(* CODESYS project Reguleringsundervisning.project

Project tree, tasks and I/O mapping:
  Device : CODESYS Control Win V3 x64, 3S - Smart Software Solutions GmbH, version 3.5.16.20
    application Application
      libraries: Standard, * (System); VisuDialogs, * (System); Util, * (System); Gand Funksjonsbibliotek, 1.1 (Gand VGS)
      task MainTask (cyclic, interval t#1ms, priority 1) calls PLC_PRG
      task ReguTask (cyclic, interval t#20ms, priority 1) calls TilbakekobletRegulering, Reguleringsprogram
      task AlarmManagerTask (cyclic, interval 50 ms, priority 31) calls AlarmManager.Alarm_Prg
      task VISU_TASK (cyclic, interval 50 ms, priority 31) calls VisuElems.Visu_Prg
      program PLC_PRG [FBD]
      Level3/
        visualisation Level3_RepOppgave_ZogN
        visualisation Level3_TilbakekobletRegulering
      TilbakekobletRegulering/
        program TilbakekobletRegulering [FBD]
        program Reguleringsprogram [FBD]
      visualisation FlytteEksempel
      global variables GVL
      Level2/
        visualisation Level2_LIC01
      Level1/
        visualisation Level1
      Level4/
        visualisation Level4_TilbakekobletRegulering_Optimalisering
      visualisation Hovedmeny
      Skogestadsmetode/
        visualisation Level3_SkogestadsMetode
        visualisation Level3_SkogestadsMetode_Nav
        visualisation Level3_SkogestadsMetode_tab1
        visualisation Level3_SkogestadsMetode_tab2
        visualisation Level3_SkogestadsMetode_tab3
        visualisation Level3_SkogestadsMetode_tab4
      FacePlates/
        visualisation Faceplate_template
        visualisation RepOppgave_FacePlate
        visualisation ZieglerNicholsSvinge1
        visualisation ZieglerNicholsSvinge2
        visualisation ZieglerNicholsSvinge3
        visualisation ZieglerNicholsSvinge4
        visualisation ZieglerNicholsSvinge5
        visualisation ZieglerNicholsSvinge6
        visualisation ZieglerNicholsSvinge7
      image pool ImagePool
      Dialogs/
        visualisation LIC01_settings
      program Belastningsim [ST]
      Symbols
      Alarm Configuration
        alarm class Error (priority 10, acknowledge REP_ACK)
        alarm class Warning (priority 30, acknowledge REP_ACK)
        alarm class Info (priority 100, acknowledge REP)
        AlarmStorage
        text list AlarmGroup1
        alarm group AlarmGroup1
            0 [Warning]: Comparison Greater, ExpressionToCompare 80, Hysteresis 5, Expression TilbakekobletRegulering.LOOP01.rPV - "Nivå høyt i vanntank"
  text list GlobalTextList
  5ce3da45-db07-42e7-a21c-a00fff4ed8f6|C:\Users\fred-olav\Pictures\Screenshots\Prosessdata.PNG
  5ce3da45-db07-42e7-a21c-a00fff4ed8f6|C:\Users\fred-olav\Pictures\Screenshots\IntProsess.PNG
  5ce3da45-db07-42e7-a21c-a00fff4ed8f6|C:\Users\Mosdal\Pictures\Formler tidskonsstant.PNG
  5ce3da45-db07-42e7-a21c-a00fff4ed8f6|C:\Users\Mosdal\Pictures\intprosess.png
  5ce3da45-db07-42e7-a21c-a00fff4ed8f6|C:\Users\Mosdal\Pictures\Formler intpros.PNG
  5ce3da45-db07-42e7-a21c-a00fff4ed8f6|C:\Users\fred-olav\Pictures\Screenshots\Formler selvregulerende.PNG
  5ce3da45-db07-42e7-a21c-a00fff4ed8f6|C:\Users\fred-olav\Pictures\Screenshots\Skjermbilde.JPG
  5ce3da45-db07-42e7-a21c-a00fff4ed8f6|C:\Users\fred-olav\Pictures\Screenshots\Formler integrerende.PNG
*)

// Device/Application/GVL
VAR_GLOBAL
	TLX:INT :=0;
	TLY:INT :=0;
	BRX:INT :=0;
	BRY:INT :=0;
	
	iSelector :INT:=1;
	
	LOOP02: Gand.Loop_CAS :=(rKp := 1.7, rTi := 10, Navn := 'LIC02', rTi_slave := 0.3);
	LOOP03: Gand.Loop_CAS := (rKp := -9.3, rTi := 15, Navn := 'Tank Nivå', rKp_slave := 0.444, rTi_slave := 2.25);
	LOOP04: Gand.Loop :=(Navn := 'Tank Nivå');
	
END_VAR

VAR_GLOBAL CONSTANT
	iMax_Pumps : INT :=10;
END_VAR

// Device/Application/PLC_PRG
PROGRAM PLC_PRG
VAR
	SP_U: BOOL;
	Verdi: REAL;
	SP: REAL;
	LLA: BOOL;
	HHA: BOOL;
	NormalShifte: REAL;
	MaxVerdi: REAL :=100;
	MinVerdi: REAL;
	HILV: REAL := 95;
	HHV: REAL :=90;
	HV: REAL := 80;
	NormalTop: REAL :=70;
	NormalBottom: REAL :=30;
	LV: REAL := 20;
	LLV: REAL :=10;
	LILV: REAL := 5;
END_VAR

// NETWORK 1

END_PROGRAM

// Device/Application/TilbakekobletRegulering/TilbakekobletRegulering
PROGRAM TilbakekobletRegulering
VAR
	Int_tids_prosess_0: Gand.Int_tids_prosess;
	Tank: Gand.Int_tids_prosess;
	LIC01: PID;
	LOOP01: Gand.Loop;
	
END_VAR
VAR_INPUT
	Belastning_LIC01: REAL :=50;
END_VAR

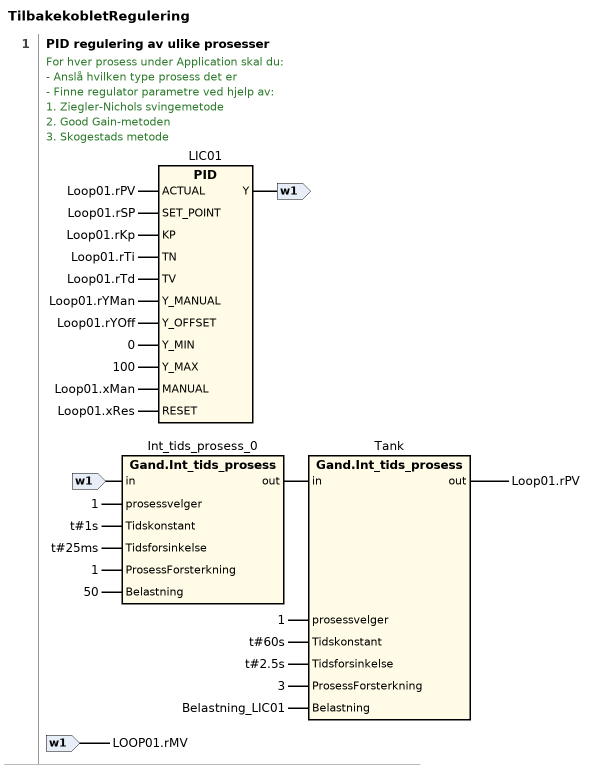
// NETWORK 1: PID regulering av ulike prosesser
// For hver prosess under Application skal du:
// - Anslå hvilken type prosess det er
// - Finne regulator parametre ved hjelp av:
// 	1. Ziegler-Nichols svingemetode
// 	2. Good Gain-metoden
// 	3. Skogestads metode
LIC01(
    ACTUAL := Loop01.rPV,
    SET_POINT := Loop01.rSP,
    KP := Loop01.rKp,
    TN := Loop01.rTi,
    TV := Loop01.rTd,
    Y_MANUAL := Loop01.rYMan,
    Y_OFFSET := Loop01.rYOff,
    Y_MIN := 0,
    Y_MAX := 100,
    MANUAL := Loop01.xMan,
    RESET := Loop01.xRes); // PID
Int_tids_prosess_0(
    in := LIC01.Y,
    prosessvelger := 1,
    Tidskonstant := t#1s,
    Tidsforsinkelse := t#25ms,
    ProsessForsterkning := 1,
    Belastning := 50); // Gand.Int_tids_prosess
Tank(
    in := Int_tids_prosess_0.out,
    prosessvelger := 1,
    Tidskonstant := t#60s,
    Tidsforsinkelse := t#2.5s,
    ProsessForsterkning := 3,
    Belastning := Belastning_LIC01); // Gand.Int_tids_prosess
Loop01.rPV := Tank.out;
LOOP01.rMV := LIC01.Y;

END_PROGRAM

// Device/Application/TilbakekobletRegulering/Reguleringsprogram
PROGRAM Reguleringsprogram
VAR
	PID01: PID;
	rSP_PID01: REAL :=50;
	rKP_PID01: REAL := 2;
	rTN_PID01: REAL := 2;
	rTV_PID01: REAL := 0;
	rYman_PID01: REAL := 20;
	rOff_PID01: REAL := 20;
	xMan_PID01: BOOL;
	xRes_PID01: BOOL;
	xLim_PID01: BOOL;
	xOvFlow_PID01: BOOL;
	Prosessnr: INT :=1;
	Prosess01: Gand.Prosess;
	
END_VAR
VAR_INPUT
	
END_VAR

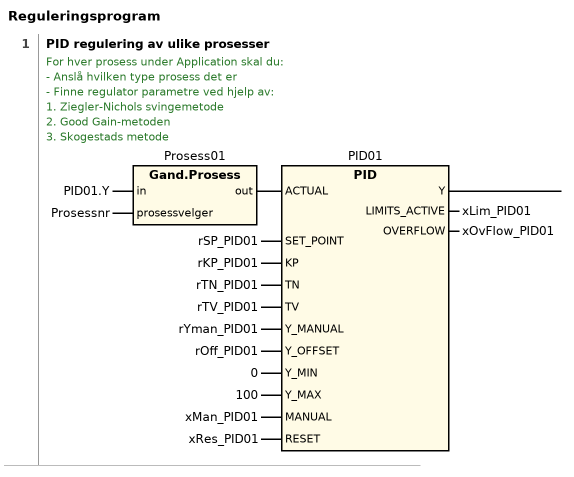
// NETWORK 1: PID regulering av ulike prosesser
// For hver prosess under Application skal du:
// - Anslå hvilken type prosess det er
// - Finne regulator parametre ved hjelp av:
// 	1. Ziegler-Nichols svingemetode
// 	2. Good Gain-metoden
// 	3. Skogestads metode
Prosess01(in := PID01.Y, prosessvelger := Prosessnr); // Gand.Prosess
PID01(
    ACTUAL := Prosess01.out,
    SET_POINT := rSP_PID01,
    KP := rKP_PID01,
    TN := rTN_PID01,
    TV := rTV_PID01,
    Y_MANUAL := rYman_PID01,
    Y_OFFSET := rOff_PID01,
    Y_MIN := 0,
    Y_MAX := 100,
    MANUAL := xMan_PID01,
    RESET := xRes_PID01,
    LIMITS_ACTIVE => xLim_PID01,
    OVERFLOW => xOvFlow_PID01); // PID

END_PROGRAM

// Device/Application/Belastningsim
PROGRAM Belastningsim
VAR
	step : INT :=1;
	i: INT;
	belastning: REAL := 50;
	timer1:TON := (PT := T#30S);
	Inntimer: BOOL :=FALSE;
END_VAR

CASE step OF
	1: 
	IF i < 100 THEN
		i:=i+1;
	ELSE
		belastning:=belastning+1;
		TilbakekobletRegulering.Belastning_LIC01:=belastning;
		i:=1;
		step:=step+1;
	END_IF
	2: 
	IF i < 100 THEN
		i:=i+1;
	ELSE
		belastning:=belastning+1;
		TilbakekobletRegulering.Belastning_LIC01:=belastning;
		i:=1;
		step:=step+1;
	END_IF
	3: 
	IF i < 100 THEN
		i:=i+1;
	ELSE
		belastning:=belastning+1;
		TilbakekobletRegulering.Belastning_LIC01:=belastning;
		i:=1;
		step:=step+1;
	END_IF
	4: 
	IF i < 100 THEN
		i:=i+1;
	ELSE
		belastning:=belastning+1;
		TilbakekobletRegulering.Belastning_LIC01:=belastning;
		i:=1;
		step:=step+1;
	END_IF
	5: 
	IF i < 100 THEN
		i:=i+1;
	ELSE
		belastning:=belastning+1;
		TilbakekobletRegulering.Belastning_LIC01:=belastning;
		i:=1;
		step:=step+1;
	END_IF
	6: 
	IF i < 100 THEN
		i:=i+1;
	ELSE
		belastning:=belastning+1;
		TilbakekobletRegulering.Belastning_LIC01:=belastning;
		i:=1;
		step:=step+1;
	END_IF
	7: 
	IF i < 100 THEN
		i:=i+1;
	ELSE
		belastning:=belastning+1;
		TilbakekobletRegulering.Belastning_LIC01:=belastning;
		i:=1;
		step:=step+1;
	END_IF
	8: 
	IF i < 100 THEN
		i:=i+1;
	ELSE
		belastning:=belastning+1;
		TilbakekobletRegulering.Belastning_LIC01:=belastning;
		i:=1;
		step:=step+1;
	END_IF
	9: 
	IF i < 100 THEN
		i:=i+1;
	ELSE
		belastning:=belastning+1;
		TilbakekobletRegulering.Belastning_LIC01:=belastning;
		i:=1;
		step:=step+1;
	END_IF
	10: 
	IF NOT Inntimer THEN
		
		IF i < 100 THEN
			i:=i+1;
		ELSE
			belastning:=belastning+1;
			TilbakekobletRegulering.Belastning_LIC01:=belastning;
			Inntimer:=TRUE;		
		END_IF
	ELSE
		IF timer1.Q THEN
		inntimer:=FALSE;
		 i:=1;
		step:=step+1;
		ELSE;
		END_IF
	END_IF
	timer1.IN:=inntimer;
	11: 
	IF i < 100 THEN
		i:=i+1;
	ELSE
		belastning:=belastning+1;
		TilbakekobletRegulering.Belastning_LIC01:=belastning;
		i:=1;
		step:=step+1;
	END_IF
	12: 
	IF i < 100 THEN
		i:=i+1;
	ELSE
		belastning:=belastning+1;
		TilbakekobletRegulering.Belastning_LIC01:=belastning;
		i:=1;
		step:=step+1;
	END_IF
	13: 
	IF i < 100 THEN
		i:=i+1;
	ELSE
		belastning:=belastning+1;
		TilbakekobletRegulering.Belastning_LIC01:=belastning;
		i:=1;
		step:=step+1;
	END_IF
	14: 
	IF i < 100 THEN
		i:=i+1;
	ELSE
		belastning:=belastning+1;
		TilbakekobletRegulering.Belastning_LIC01:=belastning;
		i:=1;
		step:=step+1;
		
	END_IF
	15: 
	IF i < 100 THEN
		i:=i+1;
	ELSE
		belastning:=belastning+1;
		TilbakekobletRegulering.Belastning_LIC01:=belastning;
		i:=1;
		step:=step+1;
	END_IF
	16: 
	IF i < 100 THEN
		i:=i+1;
	ELSE
		belastning:=belastning+1;
		TilbakekobletRegulering.Belastning_LIC01:=belastning;
		i:=1;
		step:=step+1;
	END_IF
	17: 
	IF i < 100 THEN
		i:=i+1;
	ELSE
		belastning:=belastning+1;
		TilbakekobletRegulering.Belastning_LIC01:=belastning;
		i:=1;
		step:=step+1;
	END_IF
	18: 
	IF i < 100 THEN
		i:=i+1;
	ELSE
		belastning:=belastning+1;
		TilbakekobletRegulering.Belastning_LIC01:=belastning;
		i:=1;
		step:=step+1;
	END_IF
	
END_CASE

END_PROGRAM

// Device/Application/Level4/Level4_TilbakekobletRegulering_Optimalisering
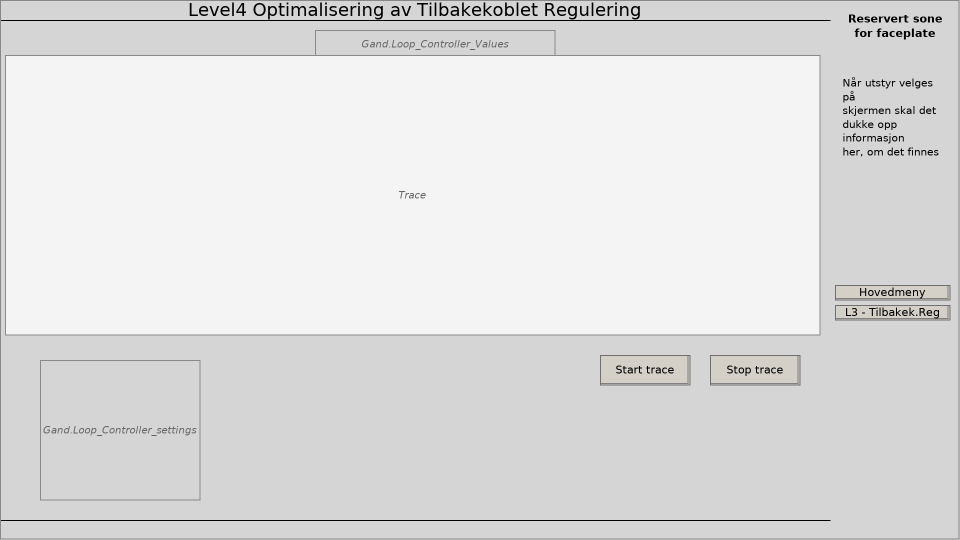
VISUALIZATION Level4_TilbakekobletRegulering_Optimalisering  // 960x540
VAR_IN_OUT
END_VAR
VAR
	bResetTrigger : BOOL;
	bStart : BOOL;
	bStop : BOOL;
	bStore : BOOL;
	sStoreFilename : STRING;
	bRestore : BOOL;
	sRestoreFilename : STRING;
END_VAR
    Frame (835,0 120x270)
        shows Faceplate_template()
        shows Navigation_template()
    Line (0,20) (830,20)
    Line (0,520) (830,520)
    Button (835,285 115x15), "Hovedmeny"
        OnMouseClick:  Assign=Hovedmeny, Type=Assignment
    Button (835,305 115x15), "L3 - Tilbakek.Reg"
        OnMouseClick:  Assign=Level3_TilbakekobletRegulering, Type=Assignment
    Label (0,0 830x20), "Level4 Optimalisering av Tilbakekoblet Regulering"
    Frame (40,360 160x140)
        shows Gand.Loop_Controller_settings(Local_data := TilbakekobletRegulering.LOOP01)
    Frame (315,30 240x28)
        shows Gand.Loop_Controller_Values(Local_data := TilbakekobletRegulering.LOOP01)
    Trace (5,55 815x280)
        p866368322: bStart
        p3851742229: bStop
    Button (600,355 90x30), "Start trace"
        toggle bStart
    Button (710,355 90x30), "Stop trace"
        toggle bStop
END_VISUALIZATION

// Device/Application/FlytteEksempel
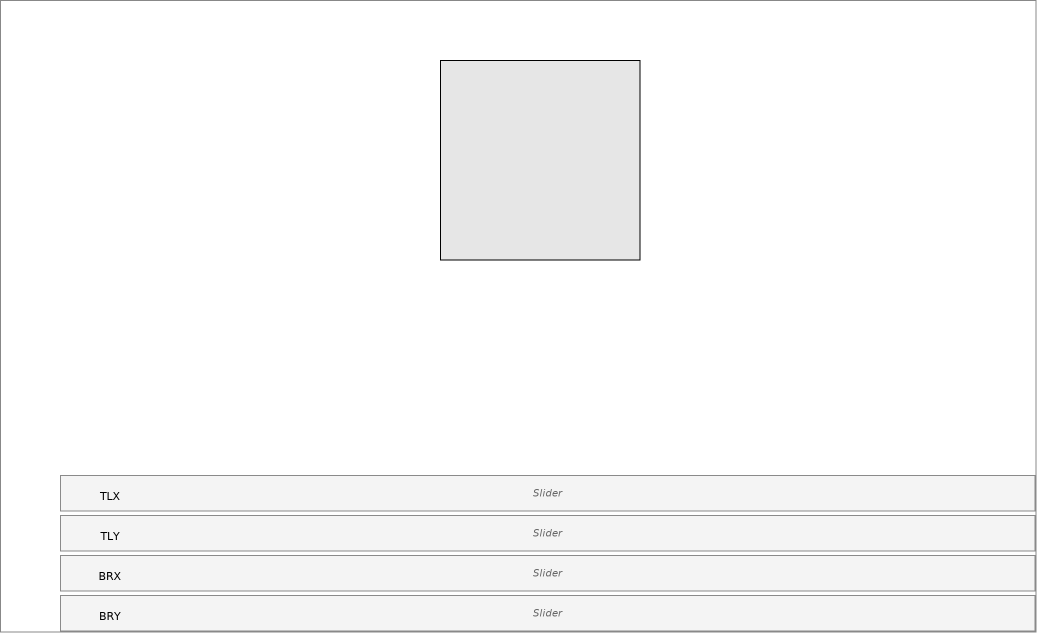
VISUALIZATION FlytteEksempel  // 1037x633
    Rectangle (440,60 200x200)
    Slider (60,475 975x36), variable: TLX, scale 0..100
    Slider (60,515 975x36), variable: TLY, scale 0..100
    Slider (60,555 975x36), variable: BRX, scale 0..100
    Slider (60,595 975x36), variable: BRY, scale 0..100
    Label (92,605 36x23), "BRY"
    Label (92,565 36x23), "BRX"
    Label (92,525 36x23), "TLY"
    Label (92,485 36x23), "TLX"
END_VISUALIZATION

// Device/Application/Level2/Level2_LIC01
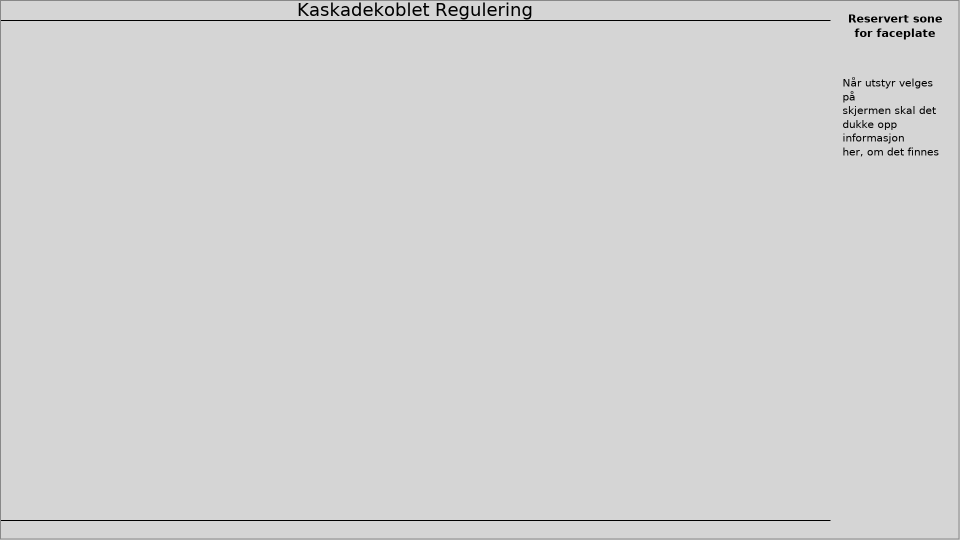
VISUALIZATION Level2_LIC01  // 960x540
VAR_IN_OUT
END_VAR
VAR
	bResetTrigger : BOOL;
	bStart : BOOL;
	bStop : BOOL;
	bStore : BOOL;
	sStoreFilename : STRING;
	bRestore : BOOL;
	sRestoreFilename : STRING;
END_VAR
    Frame (835,0 120x270)
        shows Faceplate_template()
        shows Navigation_template()
    Line (0,20) (830,20)
    Line (0,520) (830,520)
    Label (295,0 240x20), "Kaskadekoblet Regulering"
END_VISUALIZATION

// Device/Application/FacePlates/Faceplate_template
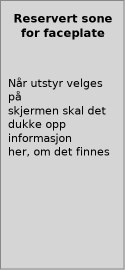
VISUALIZATION Faceplate_template  // 125x270
    Label (-12,11 150x30), "Reservert sone for faceplate"
    Label (5,75 115x85), "Når utstyr velges på skjermen skal det dukke opp informasjon her, om det finnes"
END_VISUALIZATION

// Device/Application/Hovedmeny
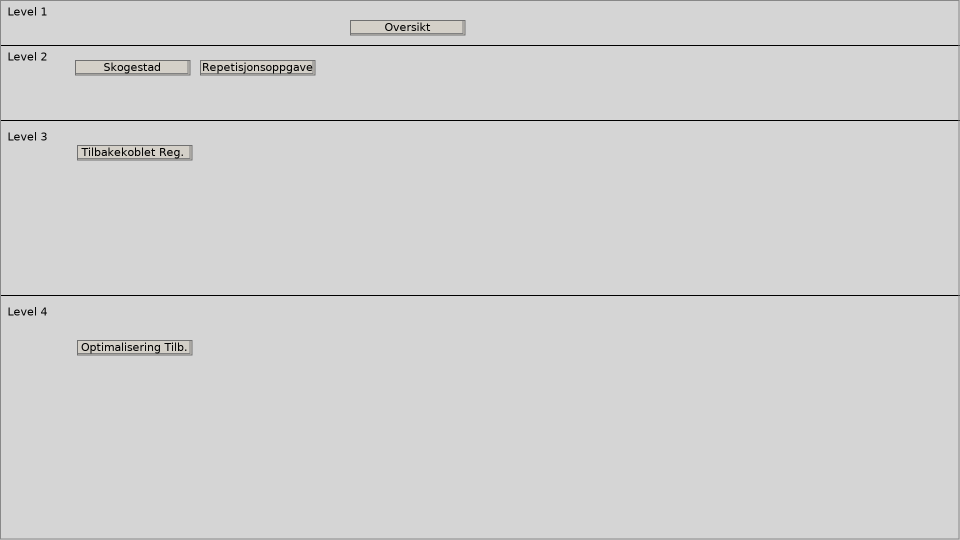
VISUALIZATION Hovedmeny  // 960x540
    Button (350,20 115x15), "Oversikt"
        OnMouseClick:  Assign=Level1, Type=Assignment
    Line (0,45) (960,45)
    Label (0,50 55x14), "Level 2"
    Label (0,130 55x14), "Level 3"
    Label (0,305 55x14), "Level 4"
    Label (0,5 55x14), "Level 1"
    Line (0,120) (960,120)
    Line (0,295) (960,295)
    Button (200,60 115x15), "Repetisjonsoppgave"
        OnMouseClick:  Assign=Level3_RepOppgave_ZogN, Type=Assignment
    Button (75,60 115x15), "Skogestad"
        OnMouseClick:  Assign=Level3_SkogestadsMetode, Type=Assignment
    Button (77,340 115x15), "Optimalisering Tilb."
        OnMouseClick:  Assign=Level4_TilbakekobletRegulering_Optimalisering, Type=Assignment
    Button (77,145 115x15), "Tilbakekoblet Reg."
        OnMouseClick:  Assign=Level3_TilbakekobletRegulering, Type=Assignment
END_VISUALIZATION

// Device/Application/Level1/Level1
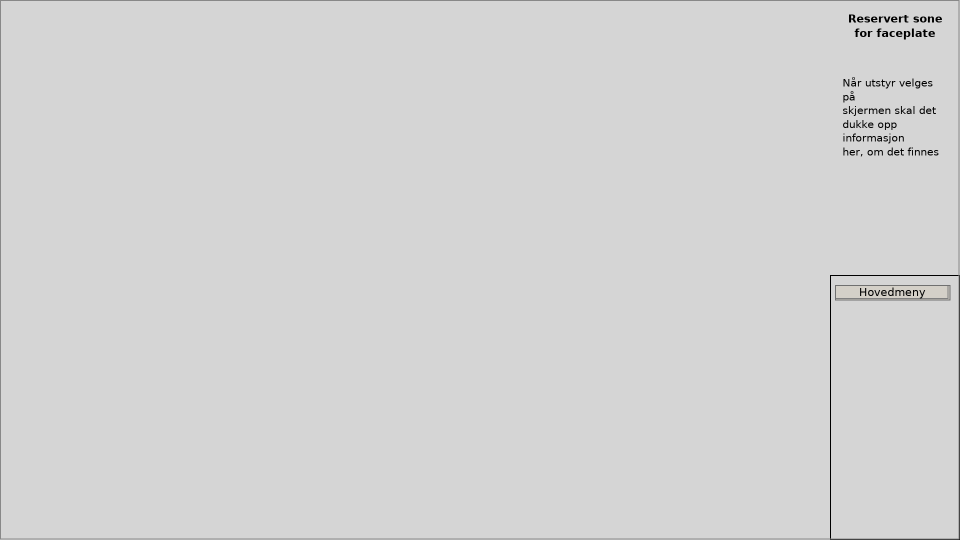
VISUALIZATION Level1  // 960x540
    Frame (835,0 120x270)
        shows Faceplate_template()
        shows Navigation_template()
    Rectangle (830,275 130x265)
    Button (835,285 115x15), "Hovedmeny"
        OnMouseClick:  Assign=Hovedmeny, Type=Assignment
END_VISUALIZATION

// Device/Application/Level3/Level3_RepOppgave_ZogN
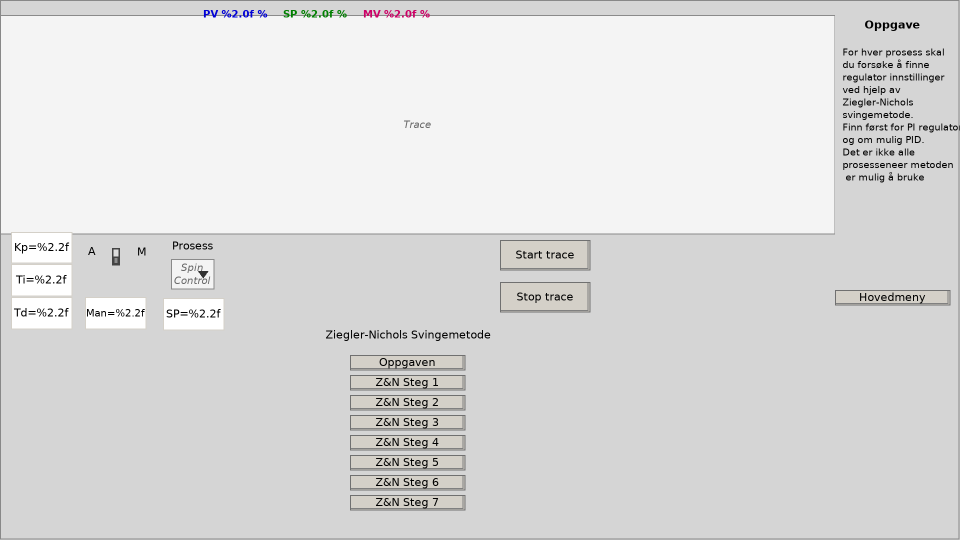
VISUALIZATION Level3_RepOppgave_ZogN  // 960x540
VAR_IN_OUT
END_VAR
VAR
	bResetTrigger : BOOL;
	bStart : BOOL;
	bStop : BOOL;
	bStore : BOOL;
	sStoreFilename : STRING;
	bRestore : BOOL;
	sRestoreFilename : STRING;
END_VAR
    Group (163,238 59x51)
        SpinControl (8,21 43x30), variable: Reguleringsprogram.Prosessnr
        Label (0,0 59x16), "Prosess"
    Trace (0,15 835x219)
        p3825648158: bResetTrigger
        p866368322: bStart
        p3851742229: bStop
        p2132035699: bStore
        p163910951: sStoreFilename
        p2217859334: bRestore
        p1301606187: sRestoreFilename
    Button (500,240 90x30), "Start trace"
        toggle bStart
    Button (500,282 90x30), "Stop trace"
        toggle bStop
    Textfield (11,232 61x31), "Kp=%2.2f", text variable: Reguleringsprogram.rKP_PID01
        OnMouseClick: write the text variable via Edit
    Textfield (11,264 61x32), "Ti=%2.2f", text variable: Reguleringsprogram.rTN_PID01
        OnMouseClick: write the text variable via Edit
    Textfield (11,297 61x32), "Td=%2.2f", text variable: Reguleringsprogram.rTV_PID01
        OnMouseClick: write the text variable via Edit
    DipSwitch (99,248 34x17), variable: Reguleringsprogram.xMan_PID01, behaviour: TOGGLE, style: Switch-DipSwitch-Gray
    Label (135,245 14x14), "M"
    Label (85,245 14x13), "A"
    Textfield (85,297 61x32), "Man=%2.2f", text variable: Reguleringsprogram.rYman_PID01
        OnMouseClick: write the text variable via Edit
    Textfield (163,298 61x32), "SP=%2.2f", text variable: Reguleringsprogram.rSP_PID01
        OnMouseClick: write the text variable via Edit
    Group (200,0 240x30)
        Textfield (0,0 80x28), "PV %2.0f %", text variable: Reguleringsprogram.PID01.ACTUAL
        Textfield (80,0 80x28), "SP %2.0f %", text variable: Reguleringsprogram.PID01.SET_POINT
        Textfield (160,0 80x28), "MV %2.0f %", text variable: Reguleringsprogram.PID01.Y
    Frame (835,0 120x270)
        shows RepOppgave_FacePlate()
        shows ZieglerNicholsSvinge1()
        shows ZieglerNicholsSvinge2()
        shows ZieglerNicholsSvinge3()
        shows ZieglerNicholsSvinge4()
        shows ZieglerNicholsSvinge5()
        shows ZieglerNicholsSvinge6()
        shows ZieglerNicholsSvinge7()
    Button (350,375 115x15), "Z&N Steg 1"
        OnMouseClick: FrameSelectionChange Selection=SelectedFrame=09a500e6-3642-417e-b93f-fcde2b0b1495, Selection=1, GlobSel=AssignType=Directly, SelType=Locally
    Button (350,395 115x15), "Z&N Steg 2"
        OnMouseClick: FrameSelectionChange Selection=SelectedFrame=09a500e6-3642-417e-b93f-fcde2b0b1495, Selection=2, GlobSel=AssignType=Directly, SelType=Locally
    Button (350,415 115x15), "Z&N Steg 3"
        OnMouseClick: FrameSelectionChange Selection=SelectedFrame=09a500e6-3642-417e-b93f-fcde2b0b1495, Selection=3, GlobSel=AssignType=Directly, SelType=Locally
    Button (350,435 115x15), "Z&N Steg 4"
        OnMouseClick: FrameSelectionChange Selection=SelectedFrame=09a500e6-3642-417e-b93f-fcde2b0b1495, Selection=4, GlobSel=AssignType=Directly, SelType=Locally
    Button (350,455 115x15), "Z&N Steg 5"
        OnMouseClick: FrameSelectionChange Selection=SelectedFrame=09a500e6-3642-417e-b93f-fcde2b0b1495, Selection=5, GlobSel=AssignType=Directly, SelType=Locally
    Button (350,475 115x15), "Z&N Steg 6"
        OnMouseClick: FrameSelectionChange Selection=SelectedFrame=09a500e6-3642-417e-b93f-fcde2b0b1495, Selection=6, GlobSel=AssignType=Directly, SelType=Locally
    Button (350,495 115x15), "Z&N Steg 7"
        OnMouseClick: FrameSelectionChange Selection=SelectedFrame=09a500e6-3642-417e-b93f-fcde2b0b1495, Selection=7, GlobSel=AssignType=Directly, SelType=Locally
    Button (350,355 115x15), "Oppgaven"
        OnMouseClick: FrameSelectionChange Selection=SelectedFrame=09a500e6-3642-417e-b93f-fcde2b0b1495, GlobSel=AssignType=Directly, SelType=Locally
    Label (315,320 187x30), "Ziegler-Nichols Svingemetode"
    Button (835,290 115x15), "Hovedmeny"
        OnMouseClick:  Assign=Hovedmeny, Type=Assignment
END_VISUALIZATION

// Device/Application/FacePlates/RepOppgave_FacePlate
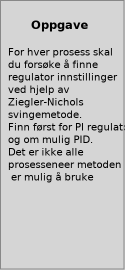
VISUALIZATION RepOppgave_FacePlate  // 125x270
    Label (20,10 80x30), "Oppgave"
    Label (5,45 110x220), "For hver prosess skal du forsøke å finne regulator innstillinger ved hjelp av Ziegler-Nichols svingemetode. Finn først for PI regulator og om mulig PID. Det er ikke alle prosesseneer metoden er mulig å bruke"
END_VISUALIZATION

// Device/Application/FacePlates/ZieglerNicholsSvinge1
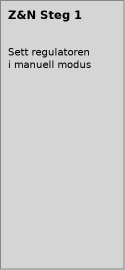
VISUALIZATION ZieglerNicholsSvinge1  // 125x270
    Label (5,0 110x30), "Z&N Steg 1"
    Label (5,45 110x220), "Sett regulatoren i manuell modus"
END_VISUALIZATION

// Device/Application/FacePlates/ZieglerNicholsSvinge2
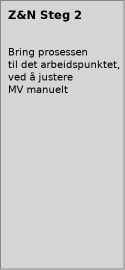
VISUALIZATION ZieglerNicholsSvinge2  // 125x270
    Label (5,0 110x30), "Z&N Steg 2"
    Label (5,45 110x220), "Bring prosessen til det arbeidspunktet, ved å justere MV manuelt"
END_VISUALIZATION

// Device/Application/FacePlates/ZieglerNicholsSvinge3
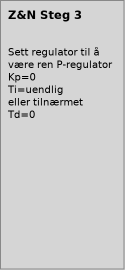
VISUALIZATION ZieglerNicholsSvinge3  // 125x270
    Label (5,0 110x30), "Z&N Steg 3"
    Label (5,45 110x220), "Sett regulator til å være ren P-regulator Kp=0 Ti=uendlig eller tilnærmet Td=0"
END_VISUALIZATION

// Device/Application/FacePlates/ZieglerNicholsSvinge4
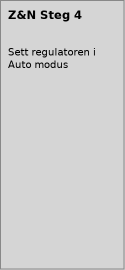
VISUALIZATION ZieglerNicholsSvinge4  // 125x270
    Label (5,0 110x30), "Z&N Steg 4"
    Label (5,45 110x220), "Sett regulatoren i Auto modus"
END_VISUALIZATION

// Device/Application/FacePlates/ZieglerNicholsSvinge5
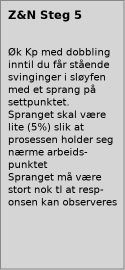
VISUALIZATION ZieglerNicholsSvinge5  // 125x270
    Label (5,0 110x30), "Z&N Steg 5"
    Label (5,45 110x220), "Øk Kp med dobbling inntil du får stående svinginger i sløyfen med et sprang på settpunktet. Spranget skal være lite (5%) slik at prosessen holder seg nærme arbeids- punktet Spranget må være stort nok tl at resp- onsen kan observeres"
END_VISUALIZATION

// Device/Application/FacePlates/ZieglerNicholsSvinge6
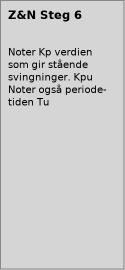
VISUALIZATION ZieglerNicholsSvinge6  // 125x270
    Label (5,0 105x30), "Z&N Steg 6"
    Label (5,45 110x220), "Noter Kp verdien som gir stående svingninger. Kpu Noter også periode- tiden Tu"
END_VISUALIZATION

// Device/Application/FacePlates/ZieglerNicholsSvinge7
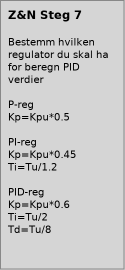
VISUALIZATION ZieglerNicholsSvinge7  // 125x270
    Label (5,0 110x30), "Z&N Steg 7"
    Label (5,35 110x235), "Bestemm hvilken regulator du skal ha for beregn PID verdier P-reg Kp=Kpu*0.5 PI-reg Kp=Kpu*0.45 Ti=Tu/1.2 PID-reg Kp=Kpu*0.6 Ti=Tu/2 Td=Tu/8"
END_VISUALIZATION

// Device/Application/Skogestadsmetode/Level3_SkogestadsMetode
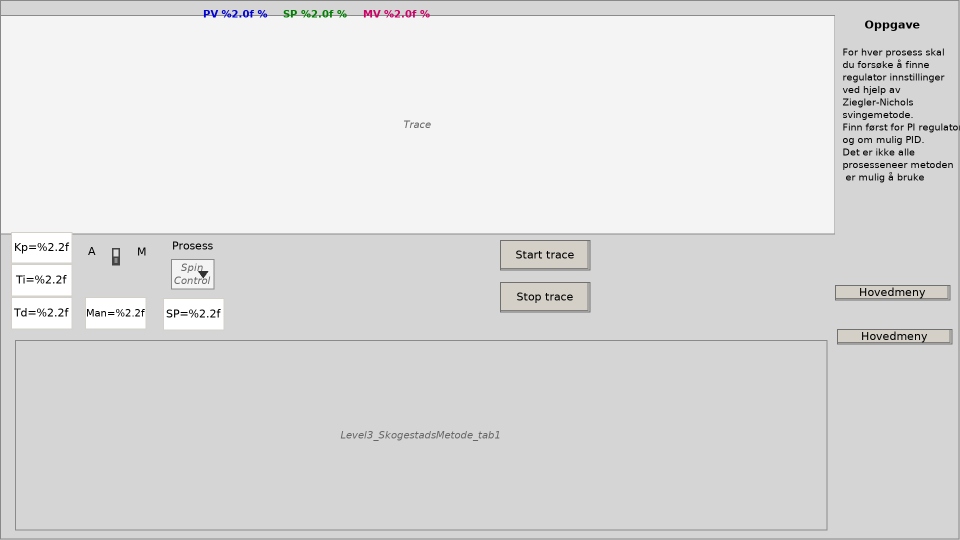
VISUALIZATION Level3_SkogestadsMetode  // 960x540
VAR_IN_OUT
END_VAR
VAR
	bResetTrigger : BOOL;
	bStart : BOOL;
	bStop : BOOL;
	bStore : BOOL;
	sStoreFilename : STRING;
	bRestore : BOOL;
	sRestoreFilename : STRING;
END_VAR
    Group (163,238 59x51)
        SpinControl (8,21 43x30), variable: Reguleringsprogram.Prosessnr
        Label (0,0 59x16), "Prosess"
    Trace (0,15 835x219)
        p3825648158: bResetTrigger
        p866368322: bStart
        p3851742229: bStop
        p2132035699: bStore
        p163910951: sStoreFilename
        p2217859334: bRestore
        p1301606187: sRestoreFilename
    Button (500,240 90x30), "Start trace"
        toggle bStart
    Button (500,282 90x30), "Stop trace"
        toggle bStop
    Textfield (11,232 61x31), "Kp=%2.2f", text variable: Reguleringsprogram.rKP_PID01
        OnMouseClick: write the text variable via Edit
    Textfield (11,264 61x32), "Ti=%2.2f", text variable: Reguleringsprogram.rTN_PID01
        OnMouseClick: write the text variable via Edit
    Textfield (11,297 61x32), "Td=%2.2f", text variable: Reguleringsprogram.rTV_PID01
        OnMouseClick: write the text variable via Edit
    DipSwitch (99,248 34x17), variable: Reguleringsprogram.xMan_PID01, behaviour: TOGGLE, style: Switch-DipSwitch-Gray
    Label (135,245 14x14), "M"
    Label (85,245 14x13), "A"
    Textfield (85,297 61x32), "Man=%2.2f", text variable: Reguleringsprogram.rYman_PID01
        OnMouseClick: write the text variable via Edit
    Textfield (163,298 61x32), "SP=%2.2f", text variable: Reguleringsprogram.rSP_PID01
        OnMouseClick: write the text variable via Edit
    Group (200,0 240x30)
        Textfield (0,0 80x28), "PV %2.0f %", text variable: Reguleringsprogram.PID01.ACTUAL
        Textfield (80,0 80x28), "SP %2.0f %", text variable: Reguleringsprogram.PID01.SET_POINT
        Textfield (160,0 80x28), "MV %2.0f %", text variable: Reguleringsprogram.PID01.Y
    Frame (835,0 120x270)
        shows RepOppgave_FacePlate()
        shows ZieglerNicholsSvinge1()
        shows ZieglerNicholsSvinge2()
        shows ZieglerNicholsSvinge3()
        shows ZieglerNicholsSvinge4()
        shows ZieglerNicholsSvinge5()
        shows ZieglerNicholsSvinge6()
        shows ZieglerNicholsSvinge7()
    TabControl (15,340 812x190)
        shows Level3_SkogestadsMetode_tab1()
        shows Level3_SkogestadsMetode_tab2()
        shows Level3_SkogestadsMetode_tab3()
        shows Level3_SkogestadsMetode_tab4()
        [0]: TabTitle=Om Skogestads Metode
        [1]: TabTitle=Integrerende vs selvstabiliserende
        [2]: TabTitle=Selvstabiliserende
        [3]: TabTitle=Integrerende prosess
    Button (835,285 115x15), "Hovedmeny"
        OnMouseClick:  Assign=Hovedmeny, Type=Assignment
    Button (837,329 115x15), "Hovedmeny"
        OnMouseClick:  Assign=Hovedmeny, Type=Assignment
END_VISUALIZATION

// Device/Application/Skogestadsmetode/Level3_SkogestadsMetode_Nav
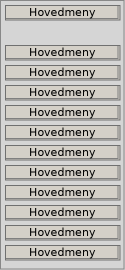
VISUALIZATION Level3_SkogestadsMetode_Nav  // 125x270
    Button (5,5 115x15), "Hovedmeny"
        OnMouseClick:  Assign=Hovedmeny, Type=Assignment
    Button (5,45 115x15), "Hovedmeny"
    Button (5,65 115x15), "Hovedmeny"
    Button (5,85 115x15), "Hovedmeny"
    Button (5,105 115x15), "Hovedmeny"
    Button (5,125 115x15), "Hovedmeny"
    Button (5,145 115x15), "Hovedmeny"
    Button (5,165 115x15), "Hovedmeny"
    Button (5,185 115x15), "Hovedmeny"
    Button (5,205 115x15), "Hovedmeny"
    Button (5,225 115x15), "Hovedmeny"
    Button (5,245 115x15), "Hovedmeny"
END_VISUALIZATION

// Device/Application/Skogestadsmetode/Level3_SkogestadsMetode_tab1
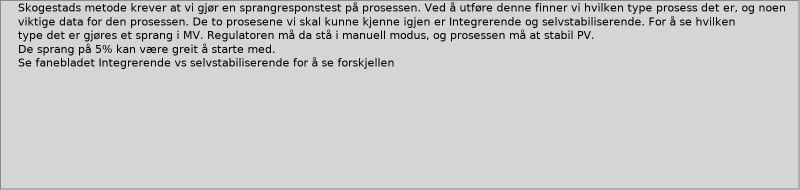
VISUALIZATION Level3_SkogestadsMetode_tab1  // 800x190
    Label (15,0 775x180), "Skogestads metode krever at vi gjør en sprangresponstest på prosessen. Ved å utføre denne finner vi hvilken type prosess det er, og noen viktige data for den prosessen. De to prosesene vi skal kunne kjenne igjen er Integrerende og selvstabiliserende. For å se hvilken type det er gjøres et sprang i MV. Regulatoren må da stå i manuell modus, og prosessen må at stabil PV. De sprang på 5% kan være greit å starte med. Se fanebladet Integrerende vs selvstabiliserende for å se forskjellen"
END_VISUALIZATION

// Device/Application/Skogestadsmetode/Level3_SkogestadsMetode_tab2
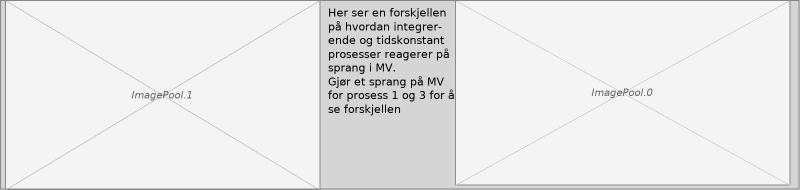
VISUALIZATION Level3_SkogestadsMetode_tab2  // 800x190
    Image (455,0 335x185), image: ImagePool.0
    Image (5,0 315x190), image: ImagePool.1
    Label (325,5 125x180), "Her ser en forskjellen på hvordan integrer- ende og tidskonstant prosesser reagerer på sprang i MV. Gjør et sprang på MV for prosess 1 og 3 for å se forskjellen"
END_VISUALIZATION

// Device/Application/Skogestadsmetode/Level3_SkogestadsMetode_tab3
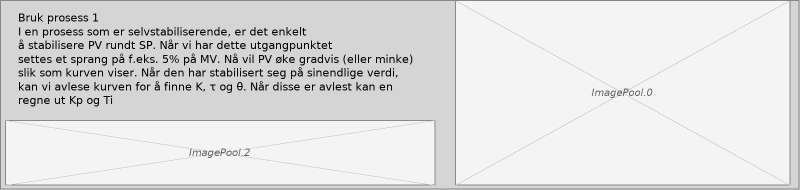
VISUALIZATION Level3_SkogestadsMetode_tab3  // 800x190
    Image (455,0 335x185), image: ImagePool.0
    Image (5,120 430x65), image: ImagePool.2
    Label (15,10 390x150), "Bruk prosess 1 I en prosess som er selvstabiliserende, er det enkelt å stabilisere PV rundt SP. Når vi har dette utgangpunktet settes et sprang på f.eks. 5% på MV. Nå vil PV øke gradvis (eller minke) slik som kurven viser. Når den har stabilisert seg på sinendlige verdi, kan vi avlese kurven for å finne K, τ og θ. Når disse er avlest kan en regne ut Kp og Ti"
END_VISUALIZATION

// Device/Application/Skogestadsmetode/Level3_SkogestadsMetode_tab4
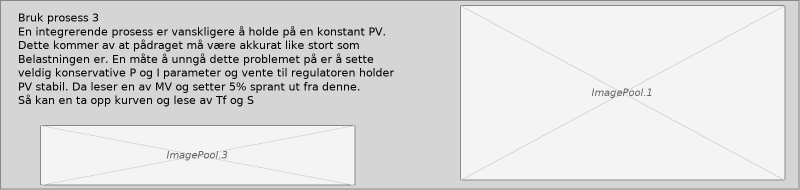
VISUALIZATION Level3_SkogestadsMetode_tab4  // 800x190
    Label (15,10 390x120), "Bruk prosess 3 En integrerende prosess er vanskligere å holde på en konstant PV. Dette kommer av at pådraget må være akkurat like stort som Belastningen er. En måte å unngå dette problemet på er å sette veldig konservative P og I parameter og vente til regulatoren holder PV stabil. Da leser en av MV og setter 5% sprant ut fra denne. Så kan en ta opp kurven og lese av Tf og S"
    Image (460,5 325x175), image: ImagePool.1
    Image (40,125 315x60), image: ImagePool.3
END_VISUALIZATION

// Device/Application/Dialogs/LIC01_settings
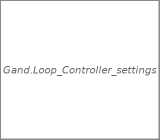
VISUALIZATION LIC01_settings  // 160x140
    Frame (0,0 160x140)
        shows Gand.Loop_Controller_settings(Local_data := TilbakekobletRegulering.LOOP01)
END_VISUALIZATION

// Device/Application/Level3/Level3_TilbakekobletRegulering
